FUNCTION_BLOCK FirstDegResponse
VAR_INPUT
	rTime:REAL;			(*Time current*)
	rDec:REAL;			(*Coeficient*)
	rInput:REAL;		(*Degree input*)
END_VAR
VAR_OUTPUT
	rOutput:REAL;
END_VAR
VAR
END_VAR

rOutput:= rInput*(1-EXPT(2.71,-rTime*rDec));

END_FUNCTION_BLOCK

(* stored: Version 1.1.0.1, ProductVersion 3.1.4024.12
   POU FirstDegResponse: Id {e874b6d4-c4a4-4ce8-9eeb-f0da9db19966}, SpecialFunc None *)
